Staubli VAL3: handleBtype.pgx

program handleBtype()
  local string l_sInputValue
begin
  // check if boolean attribute
  if (pw:sTxtBoxType[nFocused]=="B")
    if pw:sTxtBoxVal[nFocused]==pw:sTRUE
      pw:sTxtBoxVal[nFocused]=pw:sFALSE
    else
      pw:sTxtBoxVal[nFocused]="     "
      call _writeTxtBoxVal(nFocused,nVIDEONORMAL,"R")
      pw:sTxtBoxVal[nFocused]=pw:sTRUE
    endIf
    call _writeTxtBoxVal(nFocused,nVIDEOINVERSED,"R")
  else
    // If attribute is Numeric,remove 0 from string
    if (pw:sTxtBoxType[nFocused]=="N")
      // Remove 0 if present
      if pw:sTxtBoxVal[nFocused]!="0"
        call _removeChar(pw:sTxtBoxVal[nFocused],"0",1,l_sInputValue)
      else
        l_sInputValue=pw:sTxtBoxVal[nFocused]
      endIf
      call _GetUserInput(l_sInputValue)
    endIf
  endIf
end
